// TIA Portal V17 export
TagTable "Codex_Preflight_Tags"
  Sim_PreflightInt : Int  (1 s)
  Sim_PreflightReal : Real  (1 s)
